(* IEC 61131-3 sources: SRCI/RobotLibrary/Library/Constants, 3 files *)

(* ---- RobotLibraryConstants.st ---- *)
{attribute 'qualified_only'}
// -------------------------------------------------------------------------
//  SRCI Robot Library
// -------------------------------------------------------------------------
//
//  Object:      RobotLibraryConstants
//  Author:      Thorsten Brach
//  Date:        2024-06-01
//
//  Description:
//
//
//  Copyright:
//    (C) 2024 Thorsten Brach. All rights reserved
//             Licensed under the LGPL-3.0 license.
//
//  Disclaimer:
//    This project is provided without any guarantee and can be used for
//    private and commercial purposes. Any use is at the user’s
//    own risk and responsibility.
//
// -------------------------------------------------------------------------
VAR_GLOBAL CONSTANT
  /// Version of SRCI specification
  /// Bit 0-4 : Minor version = Features        (0..31)
  /// Bit 5-7 : Major version = Breaking change (0..07)
  SRCIVersion             : VersionStruct := ( MajorVersion := 1, MinorVersion := 3, PatchVersion := 0);
  /// Version of the PLC library
  PLCLibraryVersion       : VersionStruct := ( MajorVersion := 0, MinorVersion := 0, PatchVersion := 48);
  /// Minimal axes group ID
  AXES_GROUP_ID_MIN       : BYTE := 0;
  /// Maximal axes groups ID
  AXES_GROUP_ID_MAX       : BYTE := 15;
  /// OK = 0
  OK                      : DINT := 0;
  /// Running = 1
  RUNNING                 : DINT := 1;
  /// HasError = -1
  HAS_ERROR               : DINT := -1;
  /// Null pointer
  XNULL                   : DWORD := 0;
  /// Null pointer
  NULL_POINTER            : POINTER TO BYTE := 0;
  /// Real conversion factor ( REAL * 100 -> TO_INT )
  REAL_CONVERSION_FACTOR  : REAL := 100;
  /// Active command
  ACTIVE_CMD              : UDINT := 1;
  /// Buffered command
  BUFFER_CMD              : UDINT := 2;
  /// Maximal length of additional text
  MAX_ADD_TEXT_LENGTH     : DINT := 40;

  /// Minimal amount of tools
  TOOL_MIN                : DINT := 1;
  /// Minimal amount of frames
  FRAME_MIN               : DINT := 1;
  /// Minimal amount of loads
  LOAD_MIN                : DINT := 1;
  /// Minimal amount of work areas
  WORK_AREAS_MIN          : DINT := 1;
 END_VAR

(* ---- RobotLibraryDefines.st ---- *)
{attribute 'qualified_only'}
VAR_GLOBAL
  /// Count of axes groups instances
  AxesGroupInstances : BYTE;
  /// Maximal length of type name
  MaxTypeNameLength  : INT;
END_VAR

(* ---- RobotLibraryEvents.st ---- *)
{attribute 'qualified_only'}
VAR_GLOBAL
  /// Program fault : Invalid step
  ERR_INVALID_STEP             : WORD := 1;
  /// Program fault : Invalid library parameter
  ERR_INVALID_LIBRARY_PARA     : WORD := 2;
  /// Program fault : Invalid axes groups ID
  ERR_INVALID_AXES_GROUP_ID    : WORD := 3;
  /// Program fault : Invalid amount of axes groups
  ERR_INVALID_AXES_GROUP_COUNT : WORD := 4;
  /// Program fault : Timeout during command execution
  ERR_TIMEOUT_CMD              : WORD := 4;
END_VAR
